// TIA Portal V18 export
TYPE "RemConsole_IO_In"
   STRUCT
      Element_1 : Bool;
      Element_2 : Bool;
      Element_3 : Bool;
      Element_4 : Bool;
      Element_5 : Bool;
      Element_6 : Bool;
      Element_7 : Bool;
      LinkTiltRetr : Bool;
      TopDriveAux : Bool;
      LinkTiltExt : Bool;
      TopDriveEn : Bool;
      HSLTEn : Bool;
      HandlerFwd : Bool;
      HandlerRev : Bool;
      MudPumpRunning : Bool;
      QuillLock : Bool;
      BUWClose : Bool;
      BUWDown : Bool;
      BUWUp : Bool;
      TDModeMUSpin : Bool;
      TDModeMUTorq : Bool;
      TDModeRev : Bool;
      TDModeBO : Bool;
      ElevOp : Bool;
      TDExt : Bool;
      ElevCl : Bool;
      TDRet : Bool;
      PTO : Bool;
      Spare : Bool;
      MSVClose : Bool;
      MSVAuto : Bool;
      MSVOpen : Bool;
      LinkTiltFloat : Bool;
      Spare_1 : Bool;
      Spare_2 : Bool;
      Spare_3 : Bool;
      Spare_4 : Bool;
      Spare_5 : Bool;
      Heartbeat : Bool;
      Reserved : Byte;
      MUTorqLim : Int;
      DrillTorqLim : Int;
      DrillThrottle : Int;
      SpareAI : Int;
      SpareAI_1 : Int;
      SpareAI_2 : Int;
      SpareAI_3 : Int;
      SpareAI_1_1 : Int;
   END_STRUCT;
END_TYPE
